// Mitsubishi GX Works2 project: COUNTER_RST   PLC: Q03UDV

PROGRAM MAIN
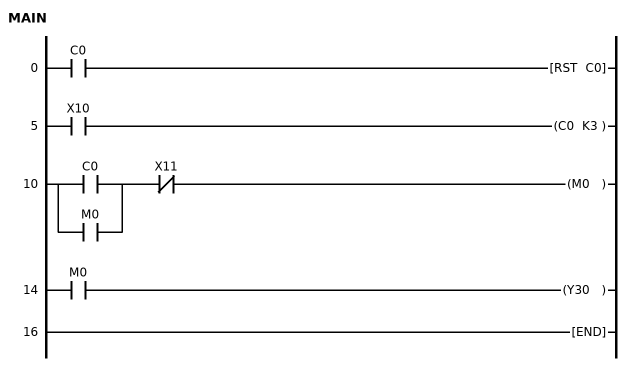
0     LD      C0
      RST     C0
5     LD      X10
      OUT     C0 K3
10    LD      C0
      OR      M0
      ANI     X11
      OUT     M0
14    LD      M0
      OUT     Y30
16    END
END_PROGRAM
